// TIA Portal V21 export
DATA_BLOCK "LifeBeatMonitor"   // DB153
{ S7_Optimized_Access := 'FALSE' }
// stored: AutoNumber false
   VAR
      CommunicationBits : Word;
      LifeBit : Bool;
      OnlineOfflineBeat : Bool;
      StartupBit : Bool;
   END_VAR
BEGIN
END_DATA_BLOCK
